FUNCTION_BLOCK ABSTRACT Insertion //IMPLEMENTS I_Insertion2D
VAR_INPUT CONSTANT
	enable : BOOL;
END_VAR
VAR_IN_OUT
	screw : EncodedDrive;
	slider : ContinuousDrive;
END_VAR
VAR_OUTPUT
	contact AT %I* : BOOL;
	home : BOOL;
	busy : BOOL;
	error : BOOL;
	
	sliderPos : LREAL;
	screwPos : LREAL;
END_VAR
(*
this abstract FB encapsulates 2 drives into a generic insertion machine
this FB cannot be used to instantiate insertions, it can only be used to refer/point to existing insertions
RETURN VALUES FOR THE METHODS ARE MEANINGLESS
*)

METHOD ABSTRACT align : BOOL
VAR_INPUT
	targetPos : REAL;
END_VAR
END_METHOD

METHOD ABSTRACT homingSequence : BOOL
VAR_INPUT
END_VAR
END_METHOD

METHOD ABSTRACT press : BOOL
VAR_INPUT
END_VAR
END_METHOD

METHOD ABSTRACT release : BOOL
VAR_INPUT
END_VAR
END_METHOD

METHOD ABSTRACT traverse : BOOL
VAR_INPUT
	direction : MC_Direction;
END_VAR
END_METHOD

END_FUNCTION_BLOCK

(* stored: Version 1.1.0.1, ProductVersion 3.1.4024.11
   POU Insertion: Id {474cec8b-539b-4b97-8920-b045f392c812}, SpecialFunc None
   Method align: Id {150b5680-ccac-4b88-b9bd-ce3a432e6e4b}
   Method homingSequence: Id {1eff6ad7-4509-4cdc-81af-eef38809ec7f}
   Method press: Id {4b68a98e-5d52-4750-8c51-39e9aab9887f}
   Method release: Id {43664641-2403-4070-8d32-2915d9eeb09e}
   Method traverse: Id {2976ba6d-a5c4-4581-84e8-a5c41da415dd} *)
